// TIA Portal V20 export
TYPE "LKinCtrl_Editor_typeHMIInterface"
// stored: Access Published
   STRUCT
      navigationWord : DWord;
      touchUp : "LKinCtrl_Editor_typeTouchUp";
      messages : "LKinCtrl_Utilities_typeMessage";
      pathEditor : "LKinCtrl_PathEditor_typeHMIInterface";
      pointEditor : "LKinCtrl_PointEditor_typeHMIInterface";
   END_STRUCT;
END_TYPE
